# EPICS autosave request: iocBoot/sioc-esb-xps1/xps.req
file xpsm.req P=ESB:XPS1:m1
file xpsm.req P=ESB:XPS1:m2
file xpsm.req P=ESB:XPS1:m3
file xpsm.req P=ESB:XPS1:m4
file xpsm.req P=ESB:XPS1:m5
file xpsm.req P=ESB:XPS1:m6
file xpsm.req P=ESB:XPS1:m7
file xpsm.req P=ESB:XPS1:m8
